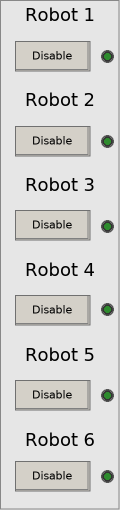
VISUALIZATION LeftRobotControls  // 120x510
    Textfield (0,0 120x30), "Robot 1"
    Textfield (0,85 120x30), "Robot 2"
    Textfield (0,170 120x30), "Robot 3"
    Textfield (0,255 120x30), "Robot 4"
        OnMouseClick: OpenDialog Dialog=VisuDialogs.MessageBox, Parameters={eType: , sMessageTxt: 'Warning Message Here', sTitle: 'WARNING'}, OpenModal=True, PositionX=312, PositionY=100
    Textfield (0,340 120x30), "Robot 5"
    Textfield (0,425 120x30), "Robot 6"
    Button (15,41 75x30), "Disable"
    Button (15,126 75x30), "Disable"
    Button (15,210 75x30), "Disable"
    Button (15,295 75x30), "Disable"
    Button (15,380 75x30), "Disable"
    Button (15,461 75x30), "Disable"
    Lamp1 (100,49 15x15), variable: TRUE, style: Lamp-Lamp1-Green
    Lamp1 (100,134 15x15), variable: TRUE, style: Lamp-Lamp1-Green
    Lamp1 (100,219 15x15), variable: TRUE, style: Lamp-Lamp1-Green
    Lamp1 (100,302 15x15), variable: TRUE, style: Lamp-Lamp1-Green
    Lamp1 (100,388 15x15), variable: TRUE, style: Lamp-Lamp1-Green
    Lamp1 (100,469 15x15), variable: TRUE, style: Lamp-Lamp1-Green
END_VISUALIZATION

(* stored: Version 1.1.0.1, ProductVersion 3.1.4024.15
   Visu LeftRobotControls: Id {9cefffad-a9dc-499d-9c0c-7d0f7528d03a} *)
